FUNCTION_BLOCK INTERNAL _StateMachine IMPLEMENTS I_Execute
VAR
	_exe					: Execute(THIS^);
	_iCurrentState			: I_StateInternal;
END_VAR

(*
Changes the current state to a new state.  

Returns:
- `Ok` - If the state transition is successful.
- `Err.Itf0` - If the new state interface is invalid.
- `None` - If the transition cannot be completed due to state conditions.
*)
METHOD Change : Result
VAR_INPUT
	iNewState	: I_StateInternal;
END_VAR
VAR_OUTPUT
	iOldState	: I_StateInternal;
END_VAR
IF iNewState = 0 THEN
	Change := Err.Itf0;
	RETURN;
END_IF

IF iNewState = _iCurrentState THEN
	Change := None;
	RETURN;
END_IF

IF NOT iNewState._CanActivate() THEN
	Change := None;
	RETURN;
END_IF

IF _iCurrentState <> 0 AND_THEN NOT _iCurrentState._CanDeactivate() THEN
	Change := None;
	RETURN;
END_IF

IF _iCurrentState <> 0 THEN
	_iCurrentState._OnExit();
END_IF

iNewState._OnEntry();
iOldState := _iCurrentState;
_iCurrentState := iNewState;
Change := Ok;
END_METHOD

METHOD Execute
VAR_INPUT
	nPhase: INT := 0;
END_VAR
IF _iCurrentState <> 0 THEN
	_iCurrentState._OnExecute();
END_IF
END_METHOD

(*
Provides access to the current state, enabling inspection or external interaction with the state.
*)
PROPERTY State : I_State
GET
State := _iCurrentState._AsIState;
END_GET
END_PROPERTY

END_FUNCTION_BLOCK

(* stored: Version 1.1.0.1
   POU _StateMachine: Id {570a94dc-a903-48df-83c5-e0703868b568}, SpecialFunc None
   Method Change: Id {c50228a6-90d0-4008-bdcd-b5914bd96cd5}
   Method Execute: Id {b879bcd6-341c-4f09-8d48-6726ba706920}
   Property State: Id {3735c750-a73c-45d9-a9dd-2c943f6399af}
   Get Get: Id {c5922222-7a05-464c-8714-df81e9760121} *)
